(* IEC 61131-3 sources: JaccoSigma/tempclass/Class/PWMJM, 1 file *)

(* ---- PWMJM.st ---- *)
(*!
<Class
	Name               = "PWMJM"
	Revision           = "0.0"
	RealtimeTask       = "true"
	DefRealtime        = "1 ms"
	CyclicTask         = "false"
	BackgroundTask     = "false"
	Sigmatek           = "false"
	OSInterface        = "false"
	HighPriority       = "false"
	Automatic          = "false"
	UpdateMode         = "Prescan"
	SharedCommandTable = "true"
	Objectsize         = "(284,120)">
	<Channels>
		<Server Name="ClassSvr" Visualized="false" Initialize="false" WriteProtected="true" Retentive="false"/>
		<Client Name="Client" Required="false" Internal="false"/>
		<Client Name="setpoint" Required="false" Internal="false"/>
	</Channels>
</Class>
*)
PWMJM : CLASS
  //Servers:
	ClassSvr 	: SvrChCmd_DINT;
  //Clients:
	Client 	: CltCh_DINT;
	setpoint 	: CltCh_DINT;
  //Variables:
		teller 	: DINT;
  //Functions:

	FUNCTION VIRTUAL GLOBAL RtWork
		VAR_INPUT
			EAX 	: UDINT;
		END_VAR
		VAR_OUTPUT
			state (EAX) 	: UDINT;
		END_VAR;
  //Tables:
	FUNCTION @STD
		VAR_OUTPUT
			ret_code	: CONFSTATES;
		END_VAR;
	FUNCTION GLOBAL TAB @CT_;
END_CLASS;

FUNCTION VIRTUAL GLOBAL PWMJM::RtWork
	VAR_INPUT
		EAX 	: UDINT;
	END_VAR
	VAR_OUTPUT
		state (EAX) 	: UDINT;
	END_VAR

  teller += 1;

  setpoint := setpoint.Read();
  if setpoint > 10 | setpoint < 0 then
    setpoint := 10;
  end_if;

  if teller >= setpoint then
    Client.Write(input:=0);
  else
    Client.Write(input:=1);
  end_if;

  if teller >= 10 then
    teller := 0;
  end_if;

 	state := READY;

END_FUNCTION
